{attribute 'GeneratedUsingTerminal: IODEVICETYPE_ETHERCATPROT'}
{attribute addProperty BoxType "IODEVICETYPE_ETHERCATPROT"}
{attribute addProperty Id "SlaveCountAT %I*UINT2DevStateAT %I*UINT2Frm0StateAT %I*UINT2Frm0WcStateAT %I*UINT2Frm0InputToggleAT %I*UINT2Frm1StateAT %I*UINT2Frm1WcStateAT %I*UINT2Frm1InputToggleAT %I*UINT2Frm2StateAT %I*UINT2Frm2WcStateAT %I*UINT2Frm2InputToggleAT %I*UINT2Frm3StateAT %I*UINT2Frm3WcStateAT %I*UINT2Frm3InputToggleAT %I*UINT2Frm4StateAT %I*UINT2Frm4WcStateAT %I*UINT2Frm4InputToggleAT %I*UINT2Frm5StateAT %I*UINT2Frm5WcStateAT %I*UINT2Frm5InputToggleAT %I*UINT2Frm6StateAT %I*UINT2Frm6WcStateAT %I*UINT2Frm6InputToggleAT %I*UINT2Frm7StateAT %I*UINT2Frm7WcStateAT %I*UINT2Frm7InputToggleAT %I*UINT2Frm8StateAT %I*UINT2Frm8WcStateAT %I*UINT2Frm8InputToggleAT %I*UINT2Frm9StateAT %I*UINT2Frm9WcStateAT %I*UINT2Frm9InputToggleAT %I*UINT2Frm10StateAT %I*UINT2Frm10WcStateAT %I*UINT2Frm10InputToggleAT %I*UINT2Frm11StateAT %I*UINT2Frm11WcStateAT %I*UINT2Frm11InputToggleAT %I*UINT2Frm12StateAT %I*UINT2Frm12WcStateAT %I*UINT2Frm12InputToggleAT %I*UINT2Frm13StateAT %I*UINT2Frm13WcStateAT %I*UINT2Frm13InputToggleAT %I*UINT2Frm14StateAT %I*UINT2Frm14WcStateAT %I*UINT2Frm14InputToggleAT %I*UINT2Frm15StateAT %I*UINT2Frm15WcStateAT %I*UINT2Frm15InputToggleAT %I*UINT2Frm16StateAT %I*UINT2Frm16WcStateAT %I*UINT2Frm16InputToggleAT %I*UINT2Frm17StateAT %I*UINT2Frm17WcStateAT %I*UINT2Frm17InputToggleAT %I*UINT2Frm18StateAT %I*UINT2Frm18WcStateAT %I*UINT2Frm18InputToggleAT %I*UINT2Frm19StateAT %I*UINT2Frm19WcStateAT %I*UINT2Frm19InputToggleAT %I*UINT2Frm20StateAT %I*UINT2Frm20WcStateAT %I*UINT2Frm20InputToggleAT %I*UINT2Frm21StateAT %I*UINT2Frm21WcStateAT %I*UINT2Frm21InputToggleAT %I*UINT2Frm22StateAT %I*UINT2Frm22WcStateAT %I*UINT2Frm22InputToggleAT %I*UINT2Frm23StateAT %I*UINT2Frm23WcStateAT %I*UINT2Frm23InputToggleAT %I*UINT2Frm24StateAT %I*UINT2Frm24WcStateAT %I*UINT2Frm24InputToggleAT %I*UINT2Frm25StateAT %I*UINT2Frm25WcStateAT %I*UINT2Frm25InputToggleAT %I*UINT2"}
{attribute addProperty CRC "631243819"}
{attribute addProperty Size "160"}
TYPE Inputs_25A0042B EXTENDS InputBase_8311D824 :
STRUCT
	{attribute addProperty Name "SlaveCount"}
	SlaveCount AT %I* : UINT;
	{attribute addProperty Name "DevState"}
	DevState AT %I* : UINT;
	{attribute addProperty Name "Frm0State"}
	Frm0State AT %I* : UINT;
	{attribute addProperty Name "Frm0WcState"}
	Frm0WcState AT %I* : UINT;
	{attribute addProperty Name "Frm0InputToggle"}
	Frm0InputToggle AT %I* : UINT;
	{attribute addProperty Name "Frm1State"}
	Frm1State AT %I* : UINT;
	{attribute addProperty Name "Frm1WcState"}
	Frm1WcState AT %I* : UINT;
	{attribute addProperty Name "Frm1InputToggle"}
	Frm1InputToggle AT %I* : UINT;
	{attribute addProperty Name "Frm2State"}
	Frm2State AT %I* : UINT;
	{attribute addProperty Name "Frm2WcState"}
	Frm2WcState AT %I* : UINT;
	{attribute addProperty Name "Frm2InputToggle"}
	Frm2InputToggle AT %I* : UINT;
	{attribute addProperty Name "Frm3State"}
	Frm3State AT %I* : UINT;
	{attribute addProperty Name "Frm3WcState"}
	Frm3WcState AT %I* : UINT;
	{attribute addProperty Name "Frm3InputToggle"}
	Frm3InputToggle AT %I* : UINT;
	{attribute addProperty Name "Frm4State"}
	Frm4State AT %I* : UINT;
	{attribute addProperty Name "Frm4WcState"}
	Frm4WcState AT %I* : UINT;
	{attribute addProperty Name "Frm4InputToggle"}
	Frm4InputToggle AT %I* : UINT;
	{attribute addProperty Name "Frm5State"}
	Frm5State AT %I* : UINT;
	{attribute addProperty Name "Frm5WcState"}
	Frm5WcState AT %I* : UINT;
	{attribute addProperty Name "Frm5InputToggle"}
	Frm5InputToggle AT %I* : UINT;
	{attribute addProperty Name "Frm6State"}
	Frm6State AT %I* : UINT;
	{attribute addProperty Name "Frm6WcState"}
	Frm6WcState AT %I* : UINT;
	{attribute addProperty Name "Frm6InputToggle"}
	Frm6InputToggle AT %I* : UINT;
	{attribute addProperty Name "Frm7State"}
	Frm7State AT %I* : UINT;
	{attribute addProperty Name "Frm7WcState"}
	Frm7WcState AT %I* : UINT;
	{attribute addProperty Name "Frm7InputToggle"}
	Frm7InputToggle AT %I* : UINT;
	{attribute addProperty Name "Frm8State"}
	Frm8State AT %I* : UINT;
	{attribute addProperty Name "Frm8WcState"}
	Frm8WcState AT %I* : UINT;
	{attribute addProperty Name "Frm8InputToggle"}
	Frm8InputToggle AT %I* : UINT;
	{attribute addProperty Name "Frm9State"}
	Frm9State AT %I* : UINT;
	{attribute addProperty Name "Frm9WcState"}
	Frm9WcState AT %I* : UINT;
	{attribute addProperty Name "Frm9InputToggle"}
	Frm9InputToggle AT %I* : UINT;
	{attribute addProperty Name "Frm10State"}
	Frm10State AT %I* : UINT;
	{attribute addProperty Name "Frm10WcState"}
	Frm10WcState AT %I* : UINT;
	{attribute addProperty Name "Frm10InputToggle"}
	Frm10InputToggle AT %I* : UINT;
	{attribute addProperty Name "Frm11State"}
	Frm11State AT %I* : UINT;
	{attribute addProperty Name "Frm11WcState"}
	Frm11WcState AT %I* : UINT;
	{attribute addProperty Name "Frm11InputToggle"}
	Frm11InputToggle AT %I* : UINT;
	{attribute addProperty Name "Frm12State"}
	Frm12State AT %I* : UINT;
	{attribute addProperty Name "Frm12WcState"}
	Frm12WcState AT %I* : UINT;
	{attribute addProperty Name "Frm12InputToggle"}
	Frm12InputToggle AT %I* : UINT;
	{attribute addProperty Name "Frm13State"}
	Frm13State AT %I* : UINT;
	{attribute addProperty Name "Frm13WcState"}
	Frm13WcState AT %I* : UINT;
	{attribute addProperty Name "Frm13InputToggle"}
	Frm13InputToggle AT %I* : UINT;
	{attribute addProperty Name "Frm14State"}
	Frm14State AT %I* : UINT;
	{attribute addProperty Name "Frm14WcState"}
	Frm14WcState AT %I* : UINT;
	{attribute addProperty Name "Frm14InputToggle"}
	Frm14InputToggle AT %I* : UINT;
	{attribute addProperty Name "Frm15State"}
	Frm15State AT %I* : UINT;
	{attribute addProperty Name "Frm15WcState"}
	Frm15WcState AT %I* : UINT;
	{attribute addProperty Name "Frm15InputToggle"}
	Frm15InputToggle AT %I* : UINT;
	{attribute addProperty Name "Frm16State"}
	Frm16State AT %I* : UINT;
	{attribute addProperty Name "Frm16WcState"}
	Frm16WcState AT %I* : UINT;
	{attribute addProperty Name "Frm16InputToggle"}
	Frm16InputToggle AT %I* : UINT;
	{attribute addProperty Name "Frm17State"}
	Frm17State AT %I* : UINT;
	{attribute addProperty Name "Frm17WcState"}
	Frm17WcState AT %I* : UINT;
	{attribute addProperty Name "Frm17InputToggle"}
	Frm17InputToggle AT %I* : UINT;
	{attribute addProperty Name "Frm18State"}
	Frm18State AT %I* : UINT;
	{attribute addProperty Name "Frm18WcState"}
	Frm18WcState AT %I* : UINT;
	{attribute addProperty Name "Frm18InputToggle"}
	Frm18InputToggle AT %I* : UINT;
	{attribute addProperty Name "Frm19State"}
	Frm19State AT %I* : UINT;
	{attribute addProperty Name "Frm19WcState"}
	Frm19WcState AT %I* : UINT;
	{attribute addProperty Name "Frm19InputToggle"}
	Frm19InputToggle AT %I* : UINT;
	{attribute addProperty Name "Frm20State"}
	Frm20State AT %I* : UINT;
	{attribute addProperty Name "Frm20WcState"}
	Frm20WcState AT %I* : UINT;
	{attribute addProperty Name "Frm20InputToggle"}
	Frm20InputToggle AT %I* : UINT;
	{attribute addProperty Name "Frm21State"}
	Frm21State AT %I* : UINT;
	{attribute addProperty Name "Frm21WcState"}
	Frm21WcState AT %I* : UINT;
	{attribute addProperty Name "Frm21InputToggle"}
	Frm21InputToggle AT %I* : UINT;
	{attribute addProperty Name "Frm22State"}
	Frm22State AT %I* : UINT;
	{attribute addProperty Name "Frm22WcState"}
	Frm22WcState AT %I* : UINT;
	{attribute addProperty Name "Frm22InputToggle"}
	Frm22InputToggle AT %I* : UINT;
	{attribute addProperty Name "Frm23State"}
	Frm23State AT %I* : UINT;
	{attribute addProperty Name "Frm23WcState"}
	Frm23WcState AT %I* : UINT;
	{attribute addProperty Name "Frm23InputToggle"}
	Frm23InputToggle AT %I* : UINT;
	{attribute addProperty Name "Frm24State"}
	Frm24State AT %I* : UINT;
	{attribute addProperty Name "Frm24WcState"}
	Frm24WcState AT %I* : UINT;
	{attribute addProperty Name "Frm24InputToggle"}
	Frm24InputToggle AT %I* : UINT;
	{attribute addProperty Name "Frm25State"}
	Frm25State AT %I* : UINT;
	{attribute addProperty Name "Frm25WcState"}
	Frm25WcState AT %I* : UINT;
	{attribute addProperty Name "Frm25InputToggle"}
	Frm25InputToggle AT %I* : UINT;
END_STRUCT
END_TYPE

(* stored: Version 1.2.0.0, ProductVersion 3.1.4024.11
   DUT Inputs_25A0042B: Id {6415fb90-d3b9-43b2-8e68-5667bfde50bd} *)
